// TIA Portal V18 export
// export: Created 2026-01-09T11:32:03.625578Z, ExportSetting WithDefaults, DisplayName Totally Integrated Automation Portal, DisplayVersion V18 Update 5, DisplayName TIA Portal Openness, DisplayVersion V18 Update 5, DisplayName TIA Portal Teamcenter Gateway, DisplayVersion V18, DisplayName TIA Portal Version Control Interface, DisplayVersion V18, DisplayName SINAMICS Startdrive Advanced, DisplayVersion V18 SP2 Update 1, DisplayName SINAMICS Startdrive G110M, G120, G120C, G120D, G120P, G115D, DisplayVersion V18 SP2 Update 1, DisplayName SINAMICS Startdrive G130, G150, S120, S150, SINAMICS MV, S210, G220, S200, DisplayVersion V18 SP2 Update 1, DisplayName STEP 7 Professional, DisplayVersion V18 Update 5, DisplayName STEP 7 Safety, DisplayVersion V18, DisplayName WinCC Professional, DisplayVersion V18 Update 5
TagTable "ST_Count"
  ST_CountClearNG : Bool  (%DB[ST_SysDBNum].DBX486.1, CPU S71500-2PN_TP700, 1 s)
  ST_CountClearOK : Bool  (%DB[ST_SysDBNum].DBX486.0, CPU S71500-2PN_TP700, 1 s)
  ST_CountClearTotal : Bool  (%DB[ST_SysDBNum].DBX486.2, CPU S71500-2PN_TP700, 1 s)
  ST_CountNG[0] : DInt  (%DB[ST_SysDBNum].DBD410, CPU S71500-2PN_TP700, 1 s)
  ST_CountNG[01] : DInt  (%DB[ST_SysDBNum].DBD414, CPU S71500-2PN_TP700, 1 s)
  ST_CountNG[02] : DInt  (%DB[ST_SysDBNum].DBD418, CPU S71500-2PN_TP700, 1 s)
  ST_CountNG[03] : DInt  (%DB[ST_SysDBNum].DBD422, CPU S71500-2PN_TP700, 1 s)
  ST_CountNG[04] : DInt  (%DB[ST_SysDBNum].DBD426, CPU S71500-2PN_TP700, 1 s)
  ST_CountNG[05] : DInt  (%DB[ST_SysDBNum].DBD430, CPU S71500-2PN_TP700, 1 s)
  ST_CountNG[06] : DInt  (%DB[ST_SysDBNum].DBD434, CPU S71500-2PN_TP700, 1 s)
  ST_CountNG[07] : DInt  (%DB[ST_SysDBNum].DBD438, CPU S71500-2PN_TP700, 1 s)
  ST_CountNG[08] : DInt  (%DB[ST_SysDBNum].DBD442, CPU S71500-2PN_TP700, 1 s)
  ST_CountNG[09] : DInt  (%DB[ST_SysDBNum].DBD446, CPU S71500-2PN_TP700, 1 s)
  ST_CountNG[10] : DInt  (%DB[ST_SysDBNum].DBD450, CPU S71500-2PN_TP700, 1 s)
  ST_CountNG[11] : DInt  (%DB[ST_SysDBNum].DBD454, CPU S71500-2PN_TP700, 1 s)
  ST_CountNG[12] : DInt  (%DB[ST_SysDBNum].DBD458, CPU S71500-2PN_TP700, 1 s)
  ST_CountNG[13] : DInt  (%DB[ST_SysDBNum].DBD462, CPU S71500-2PN_TP700, 1 s)
  ST_CountNG[14] : DInt  (%DB[ST_SysDBNum].DBD466, CPU S71500-2PN_TP700, 1 s)
  ST_CountOK[0] : DInt  (%DB[ST_SysDBNum].DBD350, CPU S71500-2PN_TP700, 1 s)
  ST_CountOK[01] : DInt  (%DB[ST_SysDBNum].DBD354, CPU S71500-2PN_TP700, 1 s)
  ST_CountOK[02] : DInt  (%DB[ST_SysDBNum].DBD358, CPU S71500-2PN_TP700, 1 s)
  ST_CountOK[03] : DInt  (%DB[ST_SysDBNum].DBD362, CPU S71500-2PN_TP700, 1 s)
  ST_CountOK[04] : DInt  (%DB[ST_SysDBNum].DBD366, CPU S71500-2PN_TP700, 1 s)
  ST_CountOK[05] : DInt  (%DB[ST_SysDBNum].DBD370, CPU S71500-2PN_TP700, 1 s)
  ST_CountOK[06] : DInt  (%DB[ST_SysDBNum].DBD374, CPU S71500-2PN_TP700, 1 s)
  ST_CountOK[07] : DInt  (%DB[ST_SysDBNum].DBD378, CPU S71500-2PN_TP700, 1 s)
  ST_CountOK[08] : DInt  (%DB[ST_SysDBNum].DBD382, CPU S71500-2PN_TP700, 1 s)
  ST_CountOK[09] : DInt  (%DB[ST_SysDBNum].DBD386, CPU S71500-2PN_TP700, 1 s)
  ST_CountOK[10] : DInt  (%DB[ST_SysDBNum].DBD390, CPU S71500-2PN_TP700, 1 s)
  ST_CountOK[11] : DInt  (%DB[ST_SysDBNum].DBD394, CPU S71500-2PN_TP700, 1 s)
  ST_CountOK[12] : DInt  (%DB[ST_SysDBNum].DBD398, CPU S71500-2PN_TP700, 1 s)
  ST_CountOK[13] : DInt  (%DB[ST_SysDBNum].DBD402, CPU S71500-2PN_TP700, 1 s)
  ST_CountOK[14] : DInt  (%DB[ST_SysDBNum].DBD406, CPU S71500-2PN_TP700, 1 s)
  ST_CountTotal : DInt  (%DB[ST_SysDBNum].DBD470, CPU S71500-2PN_TP700, 1 s)
